INTERFACE I_Button

PROPERTY IsPressed : BOOL
GET
END_GET
END_PROPERTY

END_INTERFACE

(* stored: Version 1.1.0.1, ProductVersion 3.1.4024.12
   Itf I_Button: Id {d5dd187f-5833-458e-85d4-4fcc63c344bc}
   Property IsPressed: Id {d004a021-7c3f-4b55-acca-5fc31178829d}
   Get Get: Id {7dc52437-f23f-4aff-920e-766a78346b4f} *)
